Yaskawa INFORM job: small_pipe_planes_program.JBI

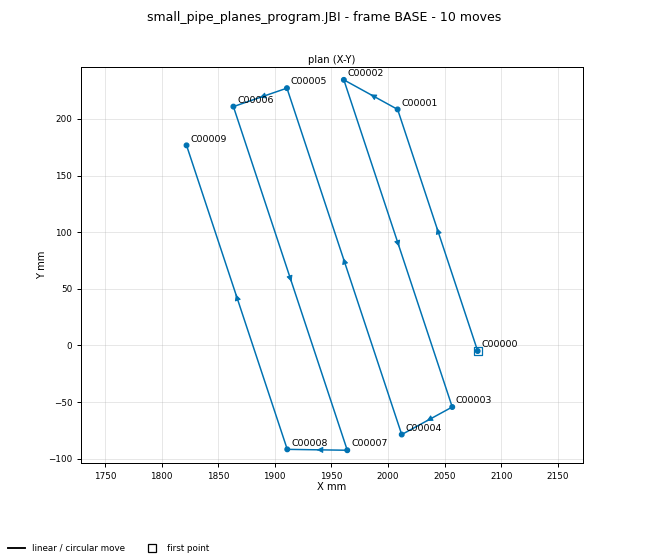
[picture p0: tool path of small_pipe_planes_program.JBI in frame BASE, 10 of 12 moves have a stored position in this frame; points joined in program order, loops and branches not executed]
/JOB
//NAME small_pipe_planes_program
//POS
///NPOS 10,0,10,0,0,0
///TOOL 0
///POSTYPE BASE
///RECTAN
///RCONF 0,0,0,0,0,0,0,0,0,0,0,0,0,0,0,0,0,0,0,0,0,0,0,0
C00000=2079.177345,-4.979739,-453.905550,175.000000,-5.000000,5.000000
C00001=2008.485272,208.370641,-455.550620,175.000000,-5.000000,5.000000
C00002=1961.007375,234.468061,-455.309620,175.000000,-5.000000,5.000000
C00003=2056.730225,-54.425807,-456.882620,175.000000,-5.000000,5.000000
C00004=2012.110324,-78.730969,-457.977620,175.000000,-5.000000,5.000000
C00005=1910.760437,227.145433,-456.884620,175.000000,-5.000000,5.000000
C00006=1863.485775,210.852404,-457.389620,175.000000,-5.000000,5.000000
C00007=1964.034092,-92.604837,-457.189620,175.000000,-5.000000,5.000000
C00008=1911.040051,-91.811507,-458.281620,175.000000,-5.000000,5.000000
C00009=1822.092763,176.633551,-457.713620,175.000000,-5.000000,5.000000
///POSTYPE PULSE
///PULSE
EC00000=18432.0
EC00001=18432.0
EC00002=18432.0
EC00003=18432.0
EC00004=18432.0
EC00005=18432.0
EC00006=18432.0
EC00007=18432.0
EC00008=18432.0
EC00009=18432.0
//INST
///DATE 2023/08/16 14:27
///ATTR SC,RW,RJ
////FRAME BASE
///GROUP1 RB1,ST1
NOP
MOVJ P009 EX000 VJ=15.00
MOVJ C00000 EC00000 VJ=15.0
CALL JOB:SPYON
MOVL C00001 EC00001 V=150.0
MOVL C00002 EC00002 V=150.0
MOVL C00003 EC00003 V=150.0
MOVL C00004 EC00004 V=150.0
MOVL C00005 EC00005 V=150.0
MOVL C00006 EC00006 V=150.0
MOVL C00007 EC00007 V=150.0
MOVL C00008 EC00008 V=150.0
MOVL C00009 EC00009 V=150.0
CALL JOB:SPYOF
MOVJ P009 VJ=15.00
END
